Fanuc KAREL source: kd00004.KL

-- PROVISIONAL review KL for V770-1; original PC SHA256 95fa042d7968ce7cebc667149c468b05a6022cccd1602fdce8af0db318417a6c
-- Incomplete behavior may be omitted. Consult companion uncertainty JSON. Do not deploy.
PROGRAM KD00004
%NOLOCKGROUP
VAR
  I : INTEGER
  J : INTEGER
  B : BOOLEAN
  R : REAL
  S : STRING[80]
BEGIN
  -- UNRESOLVED_PC offsets 5-12; opcodes 9D,23
  -- UNRESOLVED_PC offsets 17-21; opcodes 7F
END KD00004
